// TIA Portal V17 export
TagTable "Codex_Popup_PLC_Named_Int_Tags"
  DB_Components_Valve01_ClickTrig : Int  (1 s, start 0)   // Maps to DB_Components.Valve01.ClickTrig.
  DB_Components_Valve01_DoubleClickTime : Int  (1 s, start 800)   // Maps to DB_Components.Valve01.DoubleClickTime.
  DB_Components_Valve01_Switch1 : Int  (1 s, start 0)   // Maps to DB_Components.Valve01.Switch[1].
  DB_Components_Valve01_RealValue1_Int : Int  (1 s, start 0)   // Integer placeholder for DB_Components.Valve01.RealValue[1].
  DB_ActivePopup_Valve01_Visible : Int  (1 s, start 0)   // Maps to DB_ActivePopup.Valve01.Visible.
  DB_ActivePopup_Valve01_ActiveID : Int  (1 s, start 1)   // Maps to DB_ActivePopup.Valve01.ActiveID.
  DB_ActivePopup_Valve01_Confirmed : Int  (1 s, start 0)   // Maps to DB_ActivePopup.Valve01.Confirmed.
  DB_ActivePopup_Valve01_ConfirmBtn : Int  (1 s, start 0)   // Maps to DB_ActivePopup.Valve01.ConfirmBtn.
  DB_ActivePopup_Valve01_CancelBtn : Int  (1 s, start 0)   // Maps to DB_ActivePopup.Valve01.CancelBtn.
  DB_Components_Heater01_ClickTrig : Int  (1 s, start 0)   // Maps to DB_Components.Heater01.ClickTrig.
  DB_Components_Heater01_DoubleClickTime : Int  (1 s, start 800)   // Maps to DB_Components.Heater01.DoubleClickTime.
  DB_Components_Heater01_Switch1 : Int  (1 s, start 0)   // Maps to DB_Components.Heater01.Switch[1].
  DB_Components_Heater01_RealValue1_Int : Int  (1 s, start 0)   // Integer placeholder for DB_Components.Heater01.RealValue[1].
  DB_ActivePopup_Heater01_Visible : Int  (1 s, start 0)   // Maps to DB_ActivePopup.Heater01.Visible.
  DB_ActivePopup_Heater01_Confirmed : Int  (1 s, start 0)   // Maps to DB_ActivePopup.Heater01.Confirmed.
  DB_ActivePopup_Heater01_ConfirmBtn : Int  (1 s, start 0)   // Maps to DB_ActivePopup.Heater01.ConfirmBtn.
  DB_ActivePopup_Heater01_CancelBtn : Int  (1 s, start 0)   // Maps to DB_ActivePopup.Heater01.CancelBtn.
  DB_Components_Fan01_ClickTrig : Int  (1 s, start 0)   // Maps to DB_Components.Fan01.ClickTrig.
  DB_Components_Fan01_DoubleClickTime : Int  (1 s, start 800)   // Maps to DB_Components.Fan01.DoubleClickTime.
  DB_Components_Fan01_Switch1 : Int  (1 s, start 0)   // Maps to DB_Components.Fan01.Switch[1].
  DB_Components_Fan01_RealValue1_Int : Int  (1 s, start 0)   // Integer placeholder for DB_Components.Fan01.RealValue[1].
  DB_ActivePopup_Fan01_Visible : Int  (1 s, start 0)   // Maps to DB_ActivePopup.Fan01.Visible.
  DB_ActivePopup_Fan01_ActiveID : Int  (1 s, start 3)   // Maps to DB_ActivePopup.Fan01.ActiveID.
  DB_ActivePopup_Fan01_Confirmed : Int  (1 s, start 0)   // Maps to DB_ActivePopup.Fan01.Confirmed.
  DB_ActivePopup_Fan01_ConfirmBtn : Int  (1 s, start 0)   // Maps to DB_ActivePopup.Fan01.ConfirmBtn.
  DB_ActivePopup_Fan01_CancelBtn : Int  (1 s, start 0)   // Maps to DB_ActivePopup.Fan01.CancelBtn.
